# EPICS substitutions: televac.substitutions
file televac.template
{
pattern {S, TA, DN}
	{BL4B, Chop, Televac}
}
